// SIMATIC S7-200 project (STEP 7-Micro/WIN), CPU 221 REL 01.10

ORGANIZATION_BLOCK 主程序:OB1
TITLE=程序注释
BEGIN
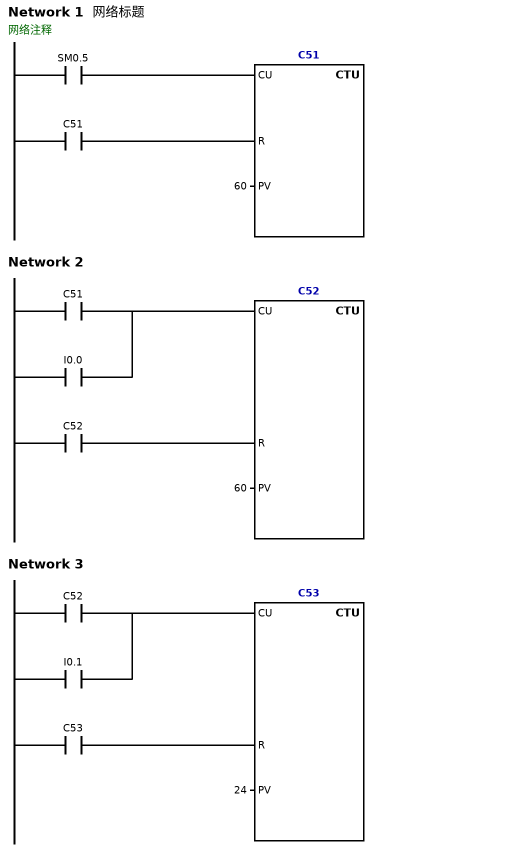
Network 1 // 网络标题
// 网络注释
LD     SM0.5
LD     C51
CTU    C51, 60
Network 2
LD     C51
O      I0.0
LD     C52
CTU    C52, 60
Network 3
LD     C52
O      I0.1
LD     C53
CTU    C53, 24
END_ORGANIZATION_BLOCK
